// TIA Portal V20 export
// export: Created 2025-12-01T14:57:32.0660167Z, ExportSetting None, DisplayName Totally Integrated Automation Portal, DisplayVersion V20 Update 3, DisplayName TIA Portal Openness, DisplayVersion V20 Update 3, DisplayName TIA Portal Version Control Interface, DisplayVersion V20 Update 3, DisplayName STEP 7 Professional, DisplayVersion V20 Update 3, DisplayName STEP 7 Safety, DisplayVersion V20 Update 2, DisplayName WinCC Basic/Comfort/Advanced, DisplayVersion V20 Update 3, DisplayName WinCC Professional, DisplayVersion V20 Update 3, DisplayName WinCC Unified, DisplayVersion V20 Update 3
DATA_BLOCK "DB885_ConfigMaquinas"   // DB885
{ S7_Optimized_Access := 'TRUE' }
// stored: AutoNumber false, MemoryReserve 0
   VAR RETAIN
      Maquina : Array[0..20] of Struct
         Nodo : UInt;   // Numero de Nodo del Variador
         DirInicial : UInt;   // Dir Inicial del Variador
         PosMaxima : Real;
         PosMinima : Real;
         NumeroDePosiciones : UInt;
         Mesa_1 : UInt;
         Mesa_2 : UInt;
         Mesa_Reposo : UInt;
         Activar_MesaReposoH2 : Bool;
         ConfigVariador : Struct
            PosicionHoming : Real;
            VelocidadHoming : Real;
            VelocidadAutomatico : Real;   // Velocidad en Manual
            ACC : Real;   // Aceleracion
            DCC : Real;   // Deceleracion
         END_STRUCT;
         Mesa : Array[0..500] of "UDT_Elevador_Config";
      END_STRUCT;
   END_VAR
BEGIN
END_DATA_BLOCK
